// TIA Portal project "MVP" (V18)

(* hardware
DEVICE "S7-1200 station_1"  S7-1200 Station
   slot 0: "Rack_0"  S7-1200 Rack  Rack  V1.0
   slot 1: "PLC_1"  CPU 1214C AC/DC/Rly  6ES7 214-1BG40-0XB0  V4.5
   slot 2: "DI 16/DQ 16x24VDC_1"  6ES7 223-1BL32-0XB0  V2.0
   slot 3: "AI 8x13BIT_1"  6ES7 231-4HF32-0XB0  V2.1
*)

// ===== PLC "PLC_1"  CPU 1214C AC/DC/Rly =====

VAR_GLOBAL   // PLC tag table "Default tag table"
   "VC" AT %Q0.0 : Bool;   // Válvula on/off da entrada do sistema de compressores
   "VT" AT %Q8.1 : Bool;   // Válvula on/off da saída do tanque separador
   "VD1" AT %Q0.2 : Bool;   // Válvula on/off da linha direta (primeira)
   "VD2" AT %Q0.3 : Bool;   // Válvula on/off da linha direta (segunda)
   "C1" AT %Q0.4 : Bool;   // Compressor 1
   "C2" AT %Q0.5 : Bool;   // Compressor 2
   "C3" AT %Q0.6 : Bool;   // Compressor 3
   "LED1" AT %Q0.7 : Bool;   // LED que avisa sobre a pressão no tanque separador
   "LED2" AT %Q1.0 : Bool;   // LED que indica se há alguma operação em curso
   "LE" AT %Q1.1 : Bool;   // LED que indica o estado de Emergência
   "H" AT %Q8.0 : Bool;   // Alarme sonoro
   "BL" AT %I0.0 : Bool;   // Botão Ligar
   "BD" AT %I0.1 : Bool;   // Botão Desligar
   "BE" AT %I0.2 : Bool;   // Botão de Emergência
   "CS1" AT %I0.3 : Bool;   // Chave seletora - Saída 1
   "CS2" AT %I0.4 : Bool;   // Chave seletora - Saída 2
   "P" AT %IW112 : Int;   // Pressão no interior do tanque separador
   "PS" AT %IW114 : Int;   // Pressão na saída do conjunto de compressores
   "PN" AT %IW116 : Int;   // Pressão da linha de abastecimento (nó estendido)
   "T" AT %IW120 : Int;   // Temperatura da linha de abastecimento (nó estendido)
   "BR" AT %I0.5 : Bool;   // Botão Reset
   "BP" AT %I0.6 : Bool;   // Botão Pausa
   "PSF6" AT %IW118 : Int;   // Pressão no tanque de SF6
   "TA" AT %IW122 : Int;   // Temperatura ambiente
   "LED3" AT %Q0.1 : Bool;   // LED que indica início/fim das etapas do MS2
   "LED4" AT %Q8.2 : Bool;   // LED que indica o estado de etapa pausada
   "BU" AT %I0.7 : Bool;   // Botão Retomada (Unpause)
END_VAR

VAR_GLOBAL CONSTANT   // PLC tag table "Default tag table"
   "Pmax" : Real := 8.0;   // Pressão máxima admissível no tanque separador
   "Pmin" : Real := 2.0;   // Pressão mínima admissível no tanque separador
   "PSmax" : Real := 8.0;   // Pressão máxima admissível na saída do conjunto de compressores
   "PSmin" : Real := 2.0;   // Pressão mínima admissível na saída do conjunto de compressores
   "PNmax" : Real := 8.0;   // Pressão máxima admissível no nó estendido
   "PNmin" : Real := 2.0;   // Pressão mínima admissível no nó estendido
   "Lmin" : Real := 4.0;   // Nível mínimo da pressão no tanque separador
   "L2" : Real := 6.0;   // Nível 2 da pressão no tanque separador
   "Tlim" : Real := 4.0;   // Nível mínimo da temperatura no nó estendido
   "Tmax" : Real := 8.0;   // Temperatura máxima admissível no nó estendido
   "Tmin" : Real := 2.0;   // Temperatura mínima admissível no nó estendido
   "gamma" : Real := 0.05;   // Constante para estabelecer um intervalo ao redor de PSF6
   "beta" : Real := 0.05;   // Constante para estabelecer um intervalo ao redor de TA
   "PNlim" : Real := 3.0;   // Nível mínimo da pressão no nó estendido
END_VAR

DATA_BLOCK "Variaveis"   // DB1
{ S7_Optimized_Access := 'TRUE' }
VERSION : 0.1
   VAR
      "Valvulas ON - MS1" : Bool := false;
      n : Int := 0;
      MS1 : Bool := false;
      "Estado anterior - MS1" : Bool := false;
      "Pisca LED1" : Bool := false;
      Inadmissivel : Bool := false;
      Emergencia : Bool := false;
      "Reset delay 1" : Bool := false;
      "Decisao automatica" : Bool := false;
      "VC ON" : Bool := false;
      "Reset delay VC 1" : Bool := false;
      "Aciona compressores" : Bool := false;
      "Reset delay VC 2" : Bool := false;
      "Desliga compressores" : Bool := false;
      MS2 : Bool := false;
      "Estado anterior - MS2" : Bool := false;
      "Aciona VD2" : Bool := false;
      "Transiciona etapa" : Bool := false;
      "VD2 ON" : Bool := false;
      "Desliga VD2" : Bool := false;
      "Tempo estourado - EB" : Bool := false;
      "Tempo estourado - EC" : Bool := false;
      "EB iniciada" : Bool := false;
      "Verifica T igual TA" : Bool := false;
      "Verifica PN e PSF6" : Bool := false;
      "Estado anterior VD2" : Bool := false;
      EB : Bool := false;
      EC : Bool := false;
      "EC iniciada" : Bool := false;
      "Verifica PN e PNlim" : Bool := false;
      "Aciona VC e compressores" : Bool := false;
      "Desliga VC e compressores" : Bool := false;
      "Estado anterior VC e comp" : Bool := false;
      "VC e compressores ON" : Bool := false;
      "Pisca LED3" : Bool := false;
      "Decide etapa" : Bool := false;
      "Etapa pausada" : Bool := false;
      "Etapa retomada" : Bool := false;
      "Pausa OFF" : Bool := false;
      "Estado anterior BP" : Bool := false;
      "BP toggled" : Bool := false;
      "VD1 ON" : Bool := false;
      "Reset delay VD1 VD2 VC" : Bool := false;
      "T inadmissivel" : Bool := false;
      "Pisca LED3 aux" : Bool := false;
      "Realiza EB" : Bool := false;
      "Realiza EC" : Bool := false;
      "LED1 - Piscar" : Bool := false;
      "LED1 - Continuo" : Bool := false;
      "LED1 - Desligar" : Bool := false;
      "Nao desliga BD" : Bool := false;
      "Nao desliga BE" : Bool := false;
      "Nao desliga Inad P" : Bool := false;
      "Nao desliga Inad PS" : Bool := false;
      "Nao desliga Inad PN" : Bool := false;
      "Nao desliga Inad T" : Bool := false;
      "Estado anterior - Emergencia" : Bool := false;
      "Estado anterior - Toggle Inad P" : Bool := false;
      "Estado anterior - Toggle Inad PS" : Bool := false;
      "Estado anterior - Toggle Inad PN" : Bool := false;
      "Estado anterior - Toggle Inad T" : Bool := false;
      "Toggle Emergencia" : Bool := false;
      "Toggle Inad P" : Bool := false;
      "Toggle Inad PS" : Bool := false;
      "Toggle Inad PN" : Bool := false;
      "Toggle Inad T" : Bool := false;
      "Always False" : Bool := false;
      "Reset delay DE" : Bool := false;
      "Reset delay cautela" : Bool := false;
      "Reset delay cautela 2" : Bool := false;
      "Estado anterior - comp MS2" : Bool := false;
      "Estado anterior - desl comp MS2" : Bool := false;
      "Pisca LED2 aux" : Bool := false;
   END_VAR
BEGIN
END_DATA_BLOCK

DATA_BLOCK "Decide LED1 - DB"   // DB19
{ S7_Optimized_Access := 'TRUE' }
VERSION : 0.1
// stored: InstanceOfName Decide LED1 - FB
"Decide LED1 - FB"
BEGIN
END_DATA_BLOCK

// folder: System blocks/Program resources

DATA_BLOCK "Delay 1"   // DB2
{ S7_Optimized_Access := 'TRUE' }
AUTHOR : Simatic
FAMILY : IEC
NAME : IEC_TMR
VERSION : 1.0
// stored: InstanceOfName IEC_TIMER
"IEC_TIMER"
BEGIN
   PT := T#3S;
END_DATA_BLOCK

DATA_BLOCK "Delay VC 1"   // DB3
{ S7_Optimized_Access := 'TRUE' }
AUTHOR : Simatic
FAMILY : IEC
NAME : IEC_TMR
VERSION : 1.0
// stored: InstanceOfName IEC_TIMER
"IEC_TIMER"
BEGIN
   PT := T#5S;
END_DATA_BLOCK

DATA_BLOCK "LED1 ON"   // DB4
{ S7_Optimized_Access := 'TRUE' }
AUTHOR : Simatic
FAMILY : IEC
NAME : IEC_TMR
VERSION : 1.0
// stored: InstanceOfName IEC_TIMER
"IEC_TIMER"
BEGIN
   PT := T#1S;
END_DATA_BLOCK

DATA_BLOCK "LED1 OFF"   // DB5
{ S7_Optimized_Access := 'TRUE' }
AUTHOR : Simatic
FAMILY : IEC
NAME : IEC_TMR
VERSION : 1.0
// stored: InstanceOfName IEC_TIMER
"IEC_TIMER"
BEGIN
   PT := T#1S;
END_DATA_BLOCK

DATA_BLOCK "Reset delay 1"   // DB6
{ S7_Optimized_Access := 'TRUE' }
AUTHOR : Simatic
FAMILY : IEC
NAME : IEC_TMR
VERSION : 1.0
// stored: InstanceOfName IEC_TIMER
"IEC_TIMER"
BEGIN
   PT := T#10MS;
END_DATA_BLOCK

DATA_BLOCK "Reset delay VC 1"   // DB7
{ S7_Optimized_Access := 'TRUE' }
AUTHOR : Simatic
FAMILY : IEC
NAME : IEC_TMR
VERSION : 1.0
// stored: InstanceOfName IEC_TIMER
"IEC_TIMER"
BEGIN
   PT := T#10MS;
END_DATA_BLOCK

DATA_BLOCK "Delay VC 2"   // DB8
{ S7_Optimized_Access := 'TRUE' }
AUTHOR : Simatic
FAMILY : IEC
NAME : IEC_TMR
VERSION : 1.0
// stored: InstanceOfName IEC_TIMER
"IEC_TIMER"
BEGIN
   PT := T#5S;
END_DATA_BLOCK

DATA_BLOCK "Reset delay VC 2"   // DB9
{ S7_Optimized_Access := 'TRUE' }
AUTHOR : Simatic
FAMILY : IEC
NAME : IEC_TMR
VERSION : 1.0
// stored: InstanceOfName IEC_TIMER
"IEC_TIMER"
BEGIN
   PT := T#10MS;
END_DATA_BLOCK

DATA_BLOCK "Contagem EB"   // DB10
{ S7_Optimized_Access := 'TRUE' }
AUTHOR : Simatic
FAMILY : IEC
NAME : IEC_TMR
VERSION : 1.0
// stored: InstanceOfName IEC_TIMER
"IEC_TIMER"
BEGIN
   PT := T#20S;
END_DATA_BLOCK

DATA_BLOCK "Contagem EC"   // DB11
{ S7_Optimized_Access := 'TRUE' }
AUTHOR : Simatic
FAMILY : IEC
NAME : IEC_TMR
VERSION : 1.0
// stored: InstanceOfName IEC_TIMER
"IEC_TIMER"
BEGIN
   PT := T#20S;
END_DATA_BLOCK

DATA_BLOCK "Delay - Decisao etapa"   // DB12
{ S7_Optimized_Access := 'TRUE' }
AUTHOR : Simatic
FAMILY : IEC
NAME : IEC_TMR
VERSION : 1.0
// stored: InstanceOfName IEC_TIMER
"IEC_TIMER"
BEGIN
   PT := T#5S;
END_DATA_BLOCK

DATA_BLOCK "Reset delay DE"   // DB13
{ S7_Optimized_Access := 'TRUE' }
AUTHOR : Simatic
FAMILY : IEC
NAME : IEC_TMR
VERSION : 1.0
// stored: InstanceOfName IEC_TIMER
"IEC_TIMER"
BEGIN
   PT := T#10MS;
END_DATA_BLOCK

DATA_BLOCK "Cautela"   // DB14
{ S7_Optimized_Access := 'TRUE' }
AUTHOR : Simatic
FAMILY : IEC
NAME : IEC_TMR
VERSION : 1.0
// stored: InstanceOfName IEC_TIMER
"IEC_TIMER"
BEGIN
   PT := T#1S;
END_DATA_BLOCK

DATA_BLOCK "LED3 ON"   // DB15
{ S7_Optimized_Access := 'TRUE' }
AUTHOR : Simatic
FAMILY : IEC
NAME : IEC_TMR
VERSION : 1.0
// stored: InstanceOfName IEC_TIMER
"IEC_TIMER"
BEGIN
   PT := T#1S;
END_DATA_BLOCK

DATA_BLOCK "LED3 OFF"   // DB16
{ S7_Optimized_Access := 'TRUE' }
AUTHOR : Simatic
FAMILY : IEC
NAME : IEC_TMR
VERSION : 1.0
// stored: InstanceOfName IEC_TIMER
"IEC_TIMER"
BEGIN
   PT := T#1S;
END_DATA_BLOCK

DATA_BLOCK "Compressores OFF - Inad P"   // DB17
{ S7_Optimized_Access := 'TRUE' }
AUTHOR : Simatic
FAMILY : IEC
NAME : IEC_TMR
VERSION : 1.0
// stored: InstanceOfName IEC_TIMER
"IEC_TIMER"
BEGIN
   PT := T#3S;
END_DATA_BLOCK

DATA_BLOCK "Compressores OFF - BE"   // DB18
{ S7_Optimized_Access := 'TRUE' }
AUTHOR : Simatic
FAMILY : IEC
NAME : IEC_TMR
VERSION : 1.0
// stored: InstanceOfName IEC_TIMER
"IEC_TIMER"
BEGIN
   PT := T#3S;
END_DATA_BLOCK

DATA_BLOCK "Compressores OFF - BD"   // DB20
{ S7_Optimized_Access := 'TRUE' }
AUTHOR : Simatic
FAMILY : IEC
NAME : IEC_TMR
VERSION : 1.0
// stored: InstanceOfName IEC_TIMER
"IEC_TIMER"
BEGIN
   PT := T#3S;
END_DATA_BLOCK

DATA_BLOCK "Compressores OFF - Inad PS"   // DB21
{ S7_Optimized_Access := 'TRUE' }
AUTHOR : Simatic
FAMILY : IEC
NAME : IEC_TMR
VERSION : 1.0
// stored: InstanceOfName IEC_TIMER
"IEC_TIMER"
BEGIN
   PT := T#3S;
END_DATA_BLOCK

DATA_BLOCK "Compressores OFF - Inad PN"   // DB22
{ S7_Optimized_Access := 'TRUE' }
AUTHOR : Simatic
FAMILY : IEC
NAME : IEC_TMR
VERSION : 1.0
// stored: InstanceOfName IEC_TIMER
"IEC_TIMER"
BEGIN
   PT := T#3S;
END_DATA_BLOCK

DATA_BLOCK "Compressores OFF - Inad T"   // DB23
{ S7_Optimized_Access := 'TRUE' }
AUTHOR : Simatic
FAMILY : IEC
NAME : IEC_TMR
VERSION : 1.0
// stored: InstanceOfName IEC_TIMER
"IEC_TIMER"
BEGIN
   PT := T#3S;
END_DATA_BLOCK

DATA_BLOCK "Reset Cautela"   // DB24
{ S7_Optimized_Access := 'TRUE' }
AUTHOR : Simatic
FAMILY : IEC
NAME : IEC_TMR
VERSION : 1.0
// stored: InstanceOfName IEC_TIMER
"IEC_TIMER"
BEGIN
   PT := T#10MS;
END_DATA_BLOCK

DATA_BLOCK "Cautela 2"   // DB25
{ S7_Optimized_Access := 'TRUE' }
AUTHOR : Simatic
FAMILY : IEC
NAME : IEC_TMR
VERSION : 1.0
// stored: InstanceOfName IEC_TIMER
"IEC_TIMER"
BEGIN
   PT := T#20MS;
END_DATA_BLOCK

DATA_BLOCK "Reset Cautela 2"   // DB26
{ S7_Optimized_Access := 'TRUE' }
AUTHOR : Simatic
FAMILY : IEC
NAME : IEC_TMR
VERSION : 1.0
// stored: InstanceOfName IEC_TIMER
"IEC_TIMER"
BEGIN
   PT := T#10MS;
END_DATA_BLOCK

DATA_BLOCK "LED2 ON"   // DB27
{ S7_Optimized_Access := 'TRUE' }
AUTHOR : Simatic
FAMILY : IEC
NAME : IEC_TMR
VERSION : 1.0
// stored: InstanceOfName IEC_TIMER
"IEC_TIMER"
BEGIN
   PT := T#1S;
END_DATA_BLOCK

DATA_BLOCK "LED2 OFF"   // DB28
{ S7_Optimized_Access := 'TRUE' }
AUTHOR : Simatic
FAMILY : IEC
NAME : IEC_TMR
VERSION : 1.0
// stored: InstanceOfName IEC_TIMER
"IEC_TIMER"
BEGIN
   PT := T#1S;
END_DATA_BLOCK

// folder: (top level)

FUNCTION_BLOCK "Decide LED1 - FB"   // FB1, LAD
{ S7_Optimized_Access := 'TRUE' }
VERSION : 0.1
   VAR_INPUT
      P : Real;   // Pressão no tanque separador
   END_VAR
BEGIN

REGION Network 1 (SCL): LED que avisa sobre a pressão no tanque separador
   IF "Variaveis".MS1 = TRUE THEN
       IF #P >= "L2" THEN
           "Variaveis"."LED1 - Continuo" := TRUE;
           "Variaveis"."LED1 - Piscar" := FALSE;
           "Variaveis"."LED1 - Desligar" := FALSE;
       ELSIF #P <= "Lmin" THEN
           "Variaveis"."LED1 - Piscar" := TRUE;
           "Variaveis"."LED1 - Continuo" := FALSE;
           "Variaveis"."LED1 - Desligar" := FALSE;
       ELSE
           "Variaveis"."LED1 - Desligar" := TRUE;
           "Variaveis"."LED1 - Piscar" := FALSE;
           "Variaveis"."LED1 - Continuo" := FALSE;
       END_IF;
   ELSE
       IF #P >= "L2" THEN
           "Variaveis"."LED1 - Continuo" := TRUE;
           "Variaveis"."LED1 - Desligar" := FALSE;
       ELSE
           "Variaveis"."LED1 - Desligar" := TRUE;
           "Variaveis"."LED1 - Continuo" := FALSE;
       END_IF;
   END_IF;
END_REGION
END_FUNCTION_BLOCK

FUNCTION "Aciona valvulas - MS1" : Void   // FC1, LAD
{ S7_Optimized_Access := 'TRUE' }
VERSION : 0.1
BEGIN

REGION Network 1: Válvula on/off da entrada do sistema de compressores
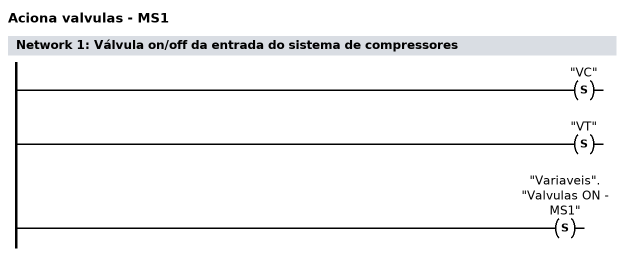
   RUNG wire#powerrail
      S_Coil( "VC" )
   END_RUNG
   RUNG wire#powerrail
      S_Coil( "VT" )
   END_RUNG
   RUNG wire#powerrail
      S_Coil( "Variaveis"."Valvulas ON - MS1" )
   END_RUNG
   // the same network as SCL:
   "VC" := TRUE;
   "VT" := TRUE;
   "Variaveis"."Valvulas ON - MS1" := TRUE;
END_REGION
END_FUNCTION

FUNCTION "Desliga valvulas - MS1" : Void   // FC2, LAD
{ S7_Optimized_Access := 'TRUE' }
VERSION : 0.1
BEGIN

REGION Network 1: Válvula on/off da entrada do sistema de compressores
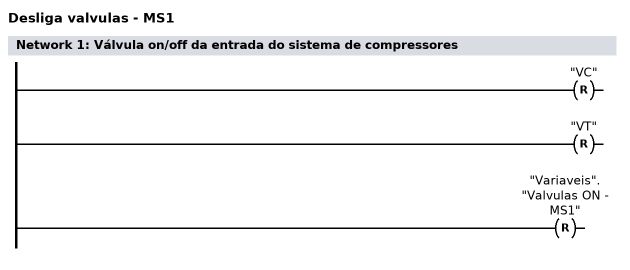
   RUNG wire#powerrail
      R_Coil( "VC" )
   END_RUNG
   RUNG wire#powerrail
      R_Coil( "VT" )
   END_RUNG
   RUNG wire#powerrail
      R_Coil( "Variaveis"."Valvulas ON - MS1" )
   END_RUNG
   // the same network as SCL:
   "VC" := FALSE;
   "VT" := FALSE;
   "Variaveis"."Valvulas ON - MS1" := FALSE;
END_REGION
END_FUNCTION

FUNCTION "Verifica valvulas 1" : Void   // FC3, LAD
{ S7_Optimized_Access := 'TRUE' }
VERSION : 0.1
BEGIN

REGION Network 1
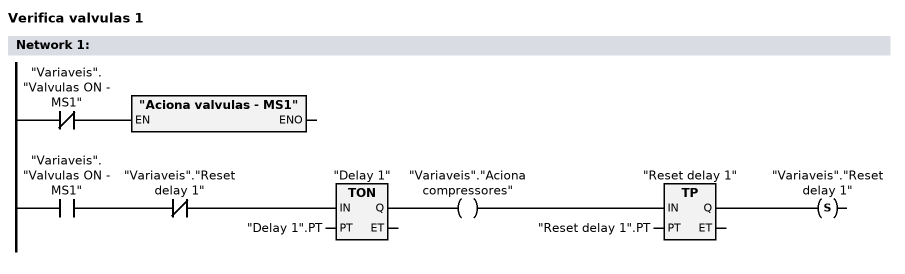
   IF NOT "Variaveis"."Valvulas ON - MS1" THEN "Aciona valvulas - MS1"(); END_IF;
   "Delay 1".TON(IN := "Variaveis"."Valvulas ON - MS1" AND NOT "Variaveis"."Reset delay 1", PT := "Delay 1".PT);
   "Variaveis"."Aciona compressores" := "Delay 1".Q;
   "Reset delay 1".TP(IN := "Delay 1".Q, PT := "Reset delay 1".PT);
   IF "Reset delay 1".Q THEN "Variaveis"."Reset delay 1" := TRUE; END_IF;
END_REGION
END_FUNCTION

FUNCTION "Verifica valvulas 2" : Void   // FC4, LAD
{ S7_Optimized_Access := 'TRUE' }
VERSION : 0.1
BEGIN

REGION Network 1
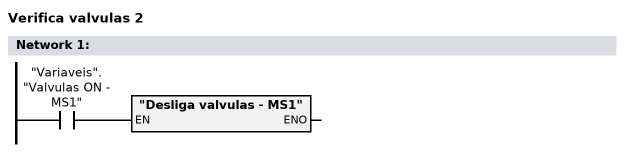
   RUNG wire#powerrail
      Contact( "Variaveis"."Valvulas ON - MS1" )
      "Desliga valvulas - MS1"()
   END_RUNG
   // the same network as SCL:
   IF "Variaveis"."Valvulas ON - MS1" THEN "Desliga valvulas - MS1"(); END_IF;
END_REGION
END_FUNCTION

FUNCTION "Aciona compressores" : Void   // FC5, LAD
{ S7_Optimized_Access := 'TRUE' }
VERSION : 0.1
BEGIN

REGION Network 1: Compressor 1
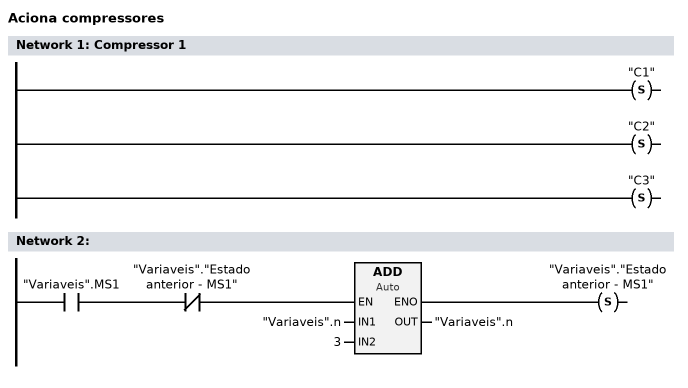
   RUNG wire#powerrail
      S_Coil( "C1" )
   END_RUNG
   RUNG wire#powerrail
      S_Coil( "C2" )
   END_RUNG
   RUNG wire#powerrail
      S_Coil( "C3" )
   END_RUNG
   // the same network as SCL:
   "C1" := TRUE;
   "C2" := TRUE;
   "C3" := TRUE;
END_REGION

REGION Network 2
   RUNG wire#powerrail
      Contact( "Variaveis".MS1 )
      I_Contact( "Variaveis"."Estado anterior - MS1" )
      Add(in1 := "Variaveis".n, in2 := 3, out => "Variaveis".n)
      S_Coil( "Variaveis"."Estado anterior - MS1" )
   END_RUNG
   // the same network as SCL:
   IF "Variaveis".MS1 AND NOT "Variaveis"."Estado anterior - MS1" THEN
       "Variaveis".n := "Variaveis".n + 3;
       "Variaveis"."Estado anterior - MS1" := TRUE;
   END_IF;
END_REGION
END_FUNCTION

FUNCTION "Desliga compressores" : Void   // FC6, LAD
{ S7_Optimized_Access := 'TRUE' }
VERSION : 0.1
BEGIN

REGION Network 1: Compressor 1
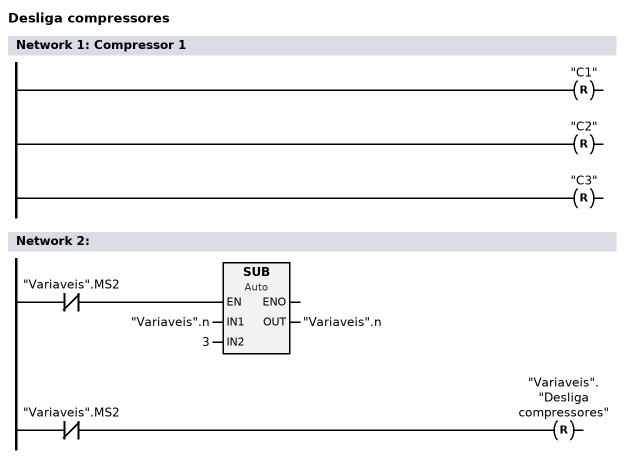
   RUNG wire#powerrail
      R_Coil( "C1" )
   END_RUNG
   RUNG wire#powerrail
      R_Coil( "C2" )
   END_RUNG
   RUNG wire#powerrail
      R_Coil( "C3" )
   END_RUNG
   // the same network as SCL:
   "C1" := FALSE;
   "C2" := FALSE;
   "C3" := FALSE;
END_REGION

REGION Network 2
   RUNG wire#powerrail
      I_Contact( "Variaveis".MS2 )
      Sub(in1 := "Variaveis".n, in2 := 3, out => "Variaveis".n)
   END_RUNG
   RUNG wire#powerrail
      I_Contact( "Variaveis".MS2 )
      R_Coil( "Variaveis"."Desliga compressores" )
   END_RUNG
   // the same network as SCL:
   IF NOT "Variaveis".MS2 THEN
       "Variaveis".n := "Variaveis".n - 3;
       "Variaveis"."Desliga compressores" := FALSE;
   END_IF;
END_REGION
END_FUNCTION

FUNCTION "Verifica compressores" : Void   // FC7, LAD
{ S7_Optimized_Access := 'TRUE' }
VERSION : 0.1
BEGIN

REGION Network 1
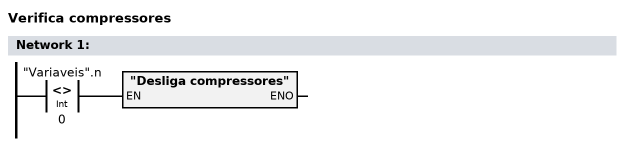
   RUNG wire#powerrail
      { S7_Templates := "SrcType := Int" } NE_Contact(in1 := "Variaveis".n, in2 := 0)
      "Desliga compressores"()
   END_RUNG
   // the same network as SCL:
   IF "Variaveis".n <> 0 THEN "Desliga compressores"(); END_IF;
END_REGION
END_FUNCTION

FUNCTION "Finaliza operacao - MS1" : Void   // FC8, LAD
{ S7_Optimized_Access := 'TRUE' }
VERSION : 0.1
BEGIN

REGION Network 1
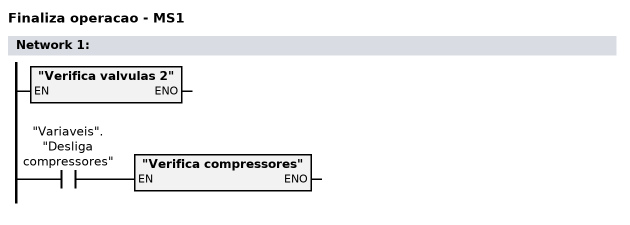
   RUNG wire#powerrail
      "Verifica valvulas 2"()
   END_RUNG
   RUNG wire#powerrail
      Contact( "Variaveis"."Desliga compressores" )
      "Verifica compressores"()
   END_RUNG
   // the same network as SCL:
   "Verifica valvulas 2"();
   IF "Variaveis"."Desliga compressores" THEN "Verifica compressores"(); END_IF;
END_REGION
END_FUNCTION

FUNCTION "MS1 - Operacao iniciada" : Void   // FC9, LAD
{ S7_Optimized_Access := 'TRUE' }
VERSION : 0.1
BEGIN

REGION Network 1
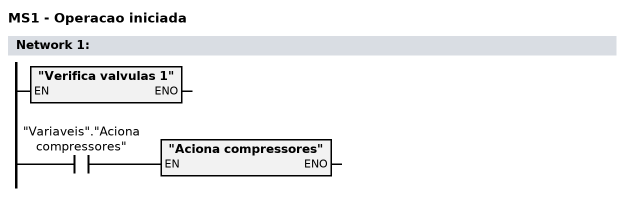
   RUNG wire#powerrail
      "Verifica valvulas 1"()
   END_RUNG
   RUNG wire#powerrail
      Contact( "Variaveis"."Aciona compressores" )
      "Aciona compressores"()
   END_RUNG
   // the same network as SCL:
   "Verifica valvulas 1"();
   IF "Variaveis"."Aciona compressores" THEN "Aciona compressores"(); END_IF;
END_REGION
END_FUNCTION

FUNCTION "MS1 - Operacao finalizada" : Void   // FC10, LAD
{ S7_Optimized_Access := 'TRUE' }
VERSION : 0.1
BEGIN

REGION Network 1
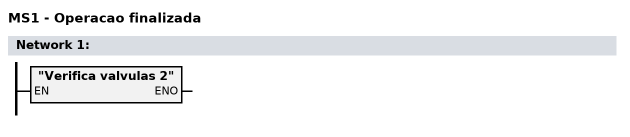
   RUNG wire#powerrail
      "Verifica valvulas 2"()
   END_RUNG
   // the same network as SCL:
   "Verifica valvulas 2"();
END_REGION
END_FUNCTION

FUNCTION "OPERACAO - MS1" : Void   // FC11, LAD
{ S7_Optimized_Access := 'TRUE' }
VERSION : 0.1
   VAR_TEMP   // added for the SCL form of the ladder/FBD networks
      _w1 : Bool;
   END_VAR
BEGIN

REGION Network 1: LED que indica se há alguma operação em curso
   // Em operação
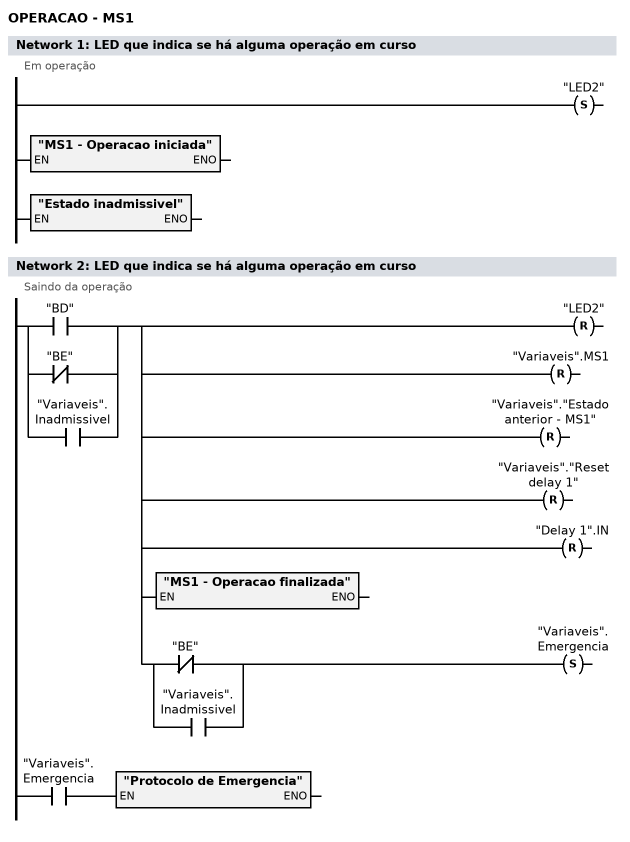
   RUNG wire#powerrail
      S_Coil( "LED2" )
   END_RUNG
   RUNG wire#powerrail
      "MS1 - Operacao iniciada"()
   END_RUNG
   RUNG wire#powerrail
      "Estado inadmissivel"()
   END_RUNG
   // the same network as SCL:
   "LED2" := TRUE;
   "MS1 - Operacao iniciada"();
   "Estado inadmissivel"();
END_REGION

REGION Network 2: LED que indica se há alguma operação em curso
   // Saindo da operação
   RUNG wire#powerrail
      Contact( "BD" )
      wire#w1
      R_Coil( "LED2" )
   END_RUNG
   RUNG wire#powerrail
      I_Contact( "BE" )
   END_RUNG wire#w1
   RUNG wire#powerrail
      Contact( "Variaveis".Inadmissivel )
   END_RUNG wire#w1
   RUNG wire#w1
      R_Coil( "Variaveis".MS1 )
   END_RUNG
   RUNG wire#w1
      R_Coil( "Variaveis"."Estado anterior - MS1" )
   END_RUNG
   RUNG wire#w1
      R_Coil( "Variaveis"."Reset delay 1" )
   END_RUNG
   RUNG wire#w1
      R_Coil( "Delay 1".IN )
   END_RUNG
   RUNG wire#w1
      "MS1 - Operacao finalizada"()
   END_RUNG
   RUNG wire#w1
      I_Contact( "BE" )
      wire#w2
      S_Coil( "Variaveis".Emergencia )
   END_RUNG
   RUNG wire#w1
      Contact( "Variaveis".Inadmissivel )
   END_RUNG wire#w2
   RUNG wire#powerrail
      Contact( "Variaveis".Emergencia )
      "Protocolo de Emergencia"()
   END_RUNG
   // the same network as SCL:
   #_w1 := "BD" OR NOT "BE" OR "Variaveis".Inadmissivel;
   IF #_w1 THEN
       "LED2" := FALSE;
       "Variaveis".MS1 := FALSE;
       "Variaveis"."Estado anterior - MS1" := FALSE;
       "Variaveis"."Reset delay 1" := FALSE;
       "Delay 1".IN := FALSE;
       "MS1 - Operacao finalizada"();
   END_IF;
   IF #_w1 AND (NOT "BE" OR "Variaveis".Inadmissivel) THEN "Variaveis".Emergencia := TRUE; END_IF;
   IF "Variaveis".Emergencia THEN "Protocolo de Emergencia"(); END_IF;
END_REGION
END_FUNCTION

FUNCTION "Pisca LED2" : Void   // FC12, LAD
{ S7_Optimized_Access := 'TRUE' }
VERSION : 0.1
   VAR_TEMP   // added for the SCL form of the ladder/FBD networks
      _w1 : Bool;
   END_VAR
BEGIN

REGION Network 1: LED que indica início/fim das etapas do MS2
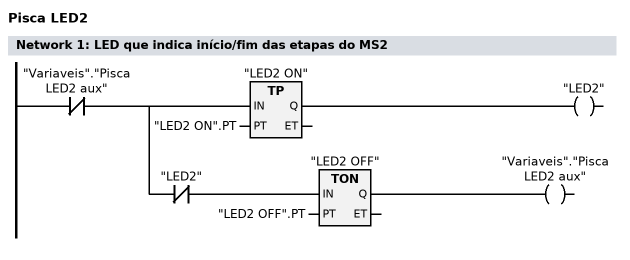
   #_w1 := NOT "Variaveis"."Pisca LED2 aux";
   "LED2 ON".TP(IN := #_w1, PT := "LED2 ON".PT);
   "LED2" := "LED2 ON".Q;
   "LED2 OFF".TON(IN := #_w1 AND NOT "LED2", PT := "LED2 OFF".PT);
   "Variaveis"."Pisca LED2 aux" := "LED2 OFF".Q;
END_REGION
END_FUNCTION

FUNCTION "Obtem pressao P" : Void   // FC13, LAD
{ S7_Optimized_Access := 'TRUE' }
VERSION : 0.1
   VAR_OUTPUT
      P : Real;   // Pressão obtida
   END_VAR
   VAR_TEMP
      "Pressao normalizada" : Real;   // Pressão normalizada
   END_VAR
BEGIN

REGION Network 1
   // Normalização do valor de pressão lido do transmissor
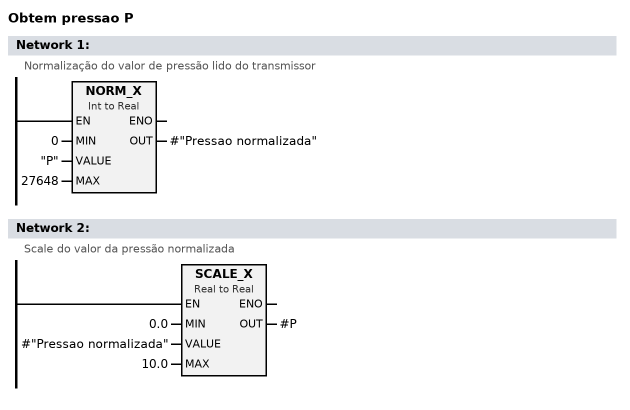
   RUNG wire#powerrail
      { S7_Templates := "[SrcType := Int, DestType := Real]" } Normalize(min := 0, value := "P", max := 27648, out => #"Pressao normalizada")
   END_RUNG
   // the same network as SCL:
   #"Pressao normalizada" := NORM_X(MIN := 0, VALUE := "P", MAX := 27648);
END_REGION

REGION Network 2
   // Scale do valor da pressão normalizada
   RUNG wire#powerrail
      { S7_Templates := "[SrcType := Real, DestType := Real]" } Scale(min := 0.0, value := #"Pressao normalizada", max := 10.0, out => #P)
   END_RUNG
   // the same network as SCL:
   #P := SCALE_X(MIN := 0.0, VALUE := #"Pressao normalizada", MAX := 10.0);
END_REGION
END_FUNCTION

FUNCTION "Estado inadmissivel" : Void   // FC14, LAD
{ S7_Optimized_Access := 'TRUE' }
VERSION : 0.1
   VAR_TEMP
      P : Real;   // Pressão P
      PS : Real;   // Pressão PS
      PN : Real;   // Pressão PN
   END_VAR
BEGIN

REGION Network 1
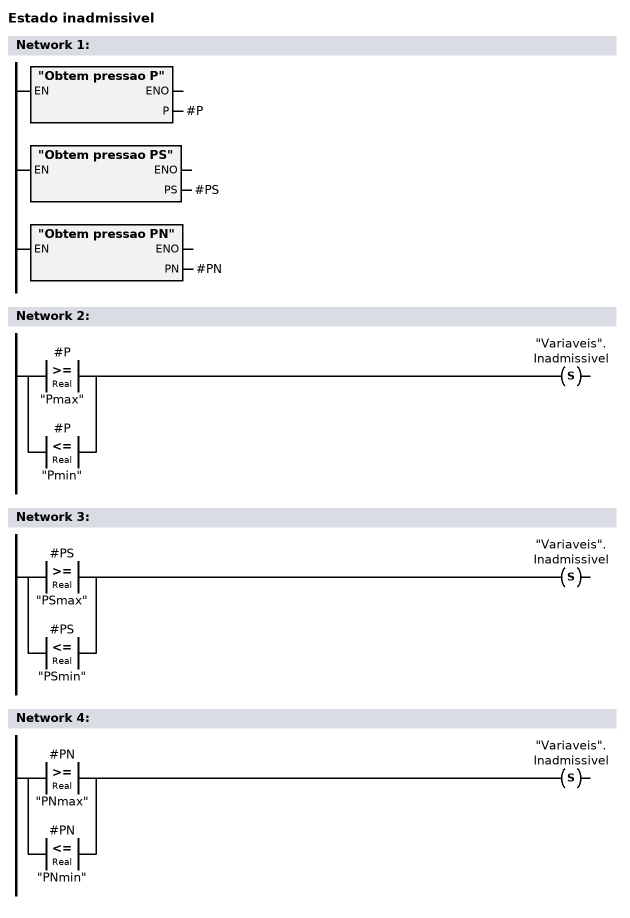
   RUNG wire#powerrail
      "Obtem pressao P"(P => #P)
   END_RUNG
   RUNG wire#powerrail
      "Obtem pressao PS"(PS => #PS)
   END_RUNG
   RUNG wire#powerrail
      "Obtem pressao PN"(PN => #PN)
   END_RUNG
   // the same network as SCL:
   "Obtem pressao P"(P => #P);
   "Obtem pressao PS"(PS => #PS);
   "Obtem pressao PN"(PN => #PN);
END_REGION

REGION Network 2
   RUNG wire#powerrail
      { S7_Templates := "SrcType := Real" } GE_Contact(in1 := #P, in2 := "Pmax")
      wire#w1
      S_Coil( "Variaveis".Inadmissivel )
   END_RUNG
   RUNG wire#powerrail
      { S7_Templates := "SrcType := Real" } LE_Contact(in1 := #P, in2 := "Pmin")
   END_RUNG wire#w1
   // the same network as SCL:
   IF (#P >= "Pmax") OR (#P <= "Pmin") THEN "Variaveis".Inadmissivel := TRUE; END_IF;
END_REGION

REGION Network 3
   RUNG wire#powerrail
      { S7_Templates := "SrcType := Real" } GE_Contact(in1 := #PS, in2 := "PSmax")
      wire#w1
      S_Coil( "Variaveis".Inadmissivel )
   END_RUNG
   RUNG wire#powerrail
      { S7_Templates := "SrcType := Real" } LE_Contact(in1 := #PS, in2 := "PSmin")
   END_RUNG wire#w1
   // the same network as SCL:
   IF (#PS >= "PSmax") OR (#PS <= "PSmin") THEN "Variaveis".Inadmissivel := TRUE; END_IF;
END_REGION

REGION Network 4
   RUNG wire#powerrail
      { S7_Templates := "SrcType := Real" } GE_Contact(in1 := #PN, in2 := "PNmax")
      wire#w1
      S_Coil( "Variaveis".Inadmissivel )
   END_RUNG
   RUNG wire#powerrail
      { S7_Templates := "SrcType := Real" } LE_Contact(in1 := #PN, in2 := "PNmin")
   END_RUNG wire#w1
   // the same network as SCL:
   IF (#PN >= "PNmax") OR (#PN <= "PNmin") THEN "Variaveis".Inadmissivel := TRUE; END_IF;
END_REGION
END_FUNCTION

FUNCTION "Obtem pressao PS" : Void   // FC15, LAD
{ S7_Optimized_Access := 'TRUE' }
VERSION : 0.1
   VAR_OUTPUT
      PS : Real;   // Pressão obtida
   END_VAR
   VAR_TEMP
      "Pressao normalizada" : Real;   // Pressão normalizada
   END_VAR
BEGIN

REGION Network 1
   // Normalização do valor de pressão lido do transmissor
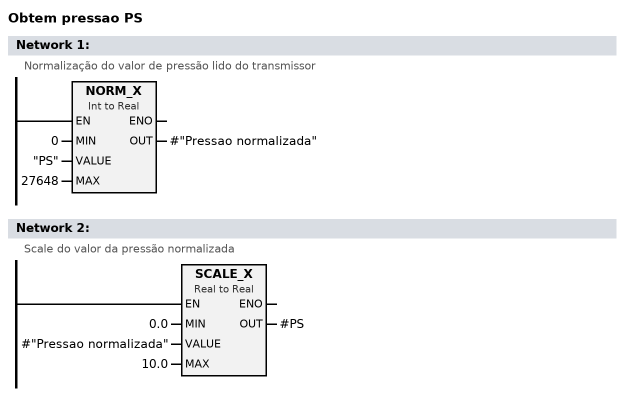
   RUNG wire#powerrail
      { S7_Templates := "[SrcType := Int, DestType := Real]" } Normalize(min := 0, value := "PS", max := 27648, out => #"Pressao normalizada")
   END_RUNG
   // the same network as SCL:
   #"Pressao normalizada" := NORM_X(MIN := 0, VALUE := "PS", MAX := 27648);
END_REGION

REGION Network 2
   // Scale do valor da pressão normalizada
   RUNG wire#powerrail
      { S7_Templates := "[SrcType := Real, DestType := Real]" } Scale(min := 0.0, value := #"Pressao normalizada", max := 10.0, out => #PS)
   END_RUNG
   // the same network as SCL:
   #PS := SCALE_X(MIN := 0.0, VALUE := #"Pressao normalizada", MAX := 10.0);
END_REGION
END_FUNCTION

FUNCTION "Obtem pressao PN" : Void   // FC16, LAD
{ S7_Optimized_Access := 'TRUE' }
VERSION : 0.1
   VAR_OUTPUT
      PN : Real;   // Pressão obtida
   END_VAR
   VAR_TEMP
      "Pressao normalizada" : Real;   // Pressão normalizada
   END_VAR
BEGIN

REGION Network 1
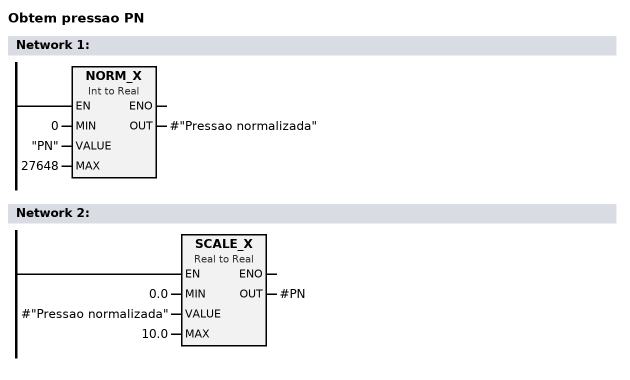
   RUNG wire#powerrail
      { S7_Templates := "[SrcType := Int, DestType := Real]" } Normalize(min := 0, value := "PN", max := 27648, out => #"Pressao normalizada")
   END_RUNG
   // the same network as SCL:
   #"Pressao normalizada" := NORM_X(MIN := 0, VALUE := "PN", MAX := 27648);
END_REGION

REGION Network 2
   RUNG wire#powerrail
      { S7_Templates := "[SrcType := Real, DestType := Real]" } Scale(min := 0.0, value := #"Pressao normalizada", max := 10.0, out => #PN)
   END_RUNG
   // the same network as SCL:
   #PN := SCALE_X(MIN := 0.0, VALUE := #"Pressao normalizada", MAX := 10.0);
END_REGION
END_FUNCTION

FUNCTION "Protocolo de Emergencia" : Void   // FC17, LAD
{ S7_Optimized_Access := 'TRUE' }
VERSION : 0.1
BEGIN

REGION Network 1: LED que indica o estado de Emergência
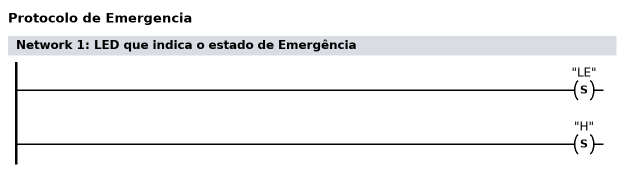
   RUNG wire#powerrail
      S_Coil( "LE" )
   END_RUNG
   RUNG wire#powerrail
      S_Coil( "H" )
   END_RUNG
   // the same network as SCL:
   "LE" := TRUE;
   "H" := TRUE;
END_REGION
END_FUNCTION

FUNCTION "Logica conjunta" : Void   // FC18, LAD
{ S7_Optimized_Access := 'TRUE' }
VERSION : 0.1
   VAR_TEMP
      P : Real;
      PS : Real;
      PN : Real;
      T : Real;
   END_VAR
BEGIN

REGION Network 1
   // Chave seletora na posição 1
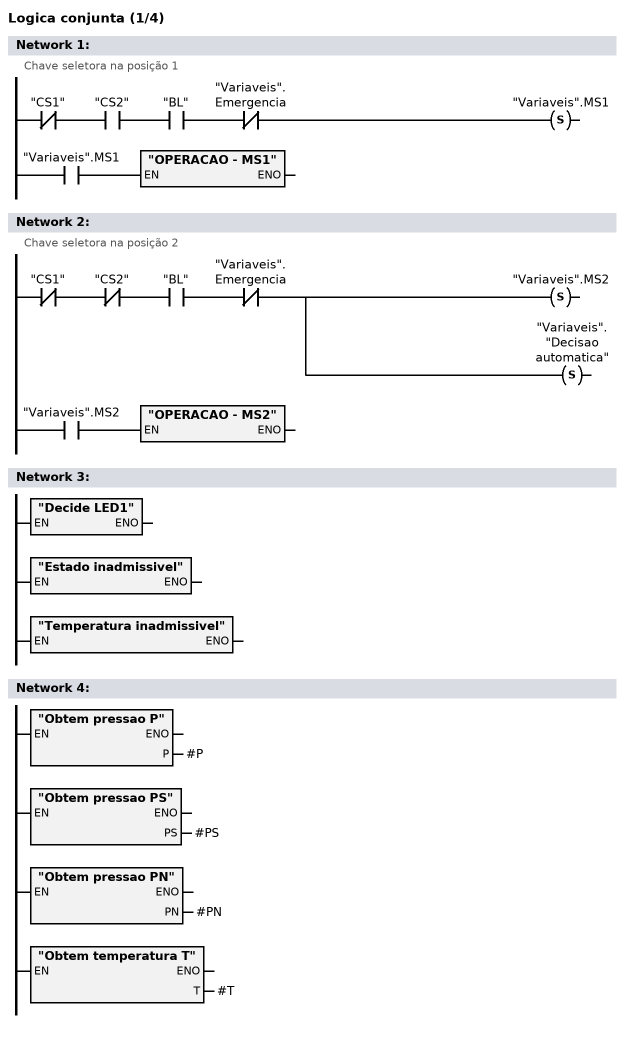
   RUNG wire#powerrail
      I_Contact( "CS1" )
      Contact( "CS2" )
      Contact( "BL" )
      I_Contact( "Variaveis".Emergencia )
      S_Coil( "Variaveis".MS1 )
   END_RUNG
   RUNG wire#powerrail
      Contact( "Variaveis".MS1 )
      "OPERACAO - MS1"()
   END_RUNG
   // the same network as SCL:
   IF NOT "CS1" AND "CS2" AND "BL" AND NOT "Variaveis".Emergencia THEN "Variaveis".MS1 := TRUE; END_IF;
   IF "Variaveis".MS1 THEN "OPERACAO - MS1"(); END_IF;
END_REGION

REGION Network 2
   // Chave seletora na posição 2
   RUNG wire#powerrail
      I_Contact( "CS1" )
      I_Contact( "CS2" )
      Contact( "BL" )
      I_Contact( "Variaveis".Emergencia )
      wire#w1
      S_Coil( "Variaveis".MS2 )
   END_RUNG
   RUNG wire#w1
      S_Coil( "Variaveis"."Decisao automatica" )
   END_RUNG
   RUNG wire#powerrail
      Contact( "Variaveis".MS2 )
      "OPERACAO - MS2"()
   END_RUNG
   // the same network as SCL:
   IF NOT "CS1" AND NOT "CS2" AND "BL" AND NOT "Variaveis".Emergencia THEN
       "Variaveis".MS2 := TRUE;
       "Variaveis"."Decisao automatica" := TRUE;
   END_IF;
   IF "Variaveis".MS2 THEN "OPERACAO - MS2"(); END_IF;
END_REGION

REGION Network 3
   RUNG wire#powerrail
      "Decide LED1"()
   END_RUNG
   RUNG wire#powerrail
      "Estado inadmissivel"()
   END_RUNG
   RUNG wire#powerrail
      "Temperatura inadmissivel"()
   END_RUNG
   // the same network as SCL:
   "Decide LED1"();
   "Estado inadmissivel"();
   "Temperatura inadmissivel"();
END_REGION

REGION Network 4
   RUNG wire#powerrail
      "Obtem pressao P"(P => #P)
   END_RUNG
   RUNG wire#powerrail
      "Obtem pressao PS"(PS => #PS)
   END_RUNG
   RUNG wire#powerrail
      "Obtem pressao PN"(PN => #PN)
   END_RUNG
   RUNG wire#powerrail
      "Obtem temperatura T"(T => #T)
   END_RUNG
   // the same network as SCL:
   "Obtem pressao P"(P => #P);
   "Obtem pressao PS"(PS => #PS);
   "Obtem pressao PN"(PN => #PN);
   "Obtem temperatura T"(T => #T);
END_REGION

REGION Network 5
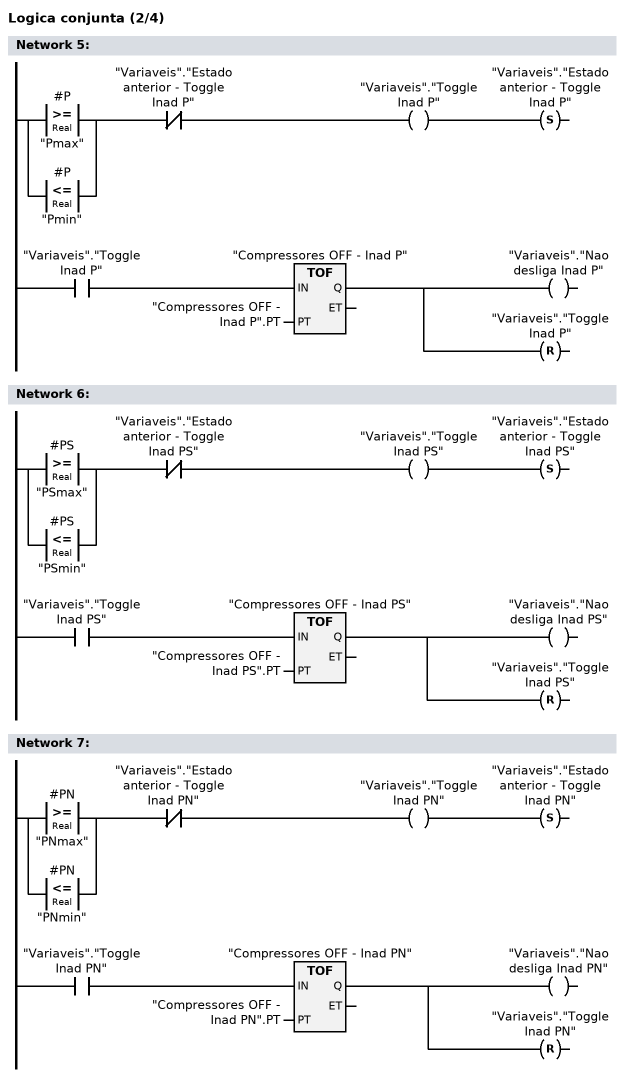
   "Variaveis"."Toggle Inad P" := ((#P >= "Pmax") OR (#P <= "Pmin")) AND NOT "Variaveis"."Estado anterior - Toggle Inad P";
   IF "Variaveis"."Toggle Inad P" THEN "Variaveis"."Estado anterior - Toggle Inad P" := TRUE; END_IF;
   "Compressores OFF - Inad P".TOF(IN := "Variaveis"."Toggle Inad P", PT := "Compressores OFF - Inad P".PT);
   "Variaveis"."Nao desliga Inad P" := "Compressores OFF - Inad P".Q;
   IF "Compressores OFF - Inad P".Q THEN "Variaveis"."Toggle Inad P" := FALSE; END_IF;
END_REGION

REGION Network 6
   "Variaveis"."Toggle Inad PS" := ((#PS >= "PSmax") OR (#PS <= "PSmin")) AND NOT "Variaveis"."Estado anterior - Toggle Inad PS";
   IF "Variaveis"."Toggle Inad PS" THEN "Variaveis"."Estado anterior - Toggle Inad PS" := TRUE; END_IF;
   "Compressores OFF - Inad PS".TOF(IN := "Variaveis"."Toggle Inad PS", PT := "Compressores OFF - Inad PS".PT);
   "Variaveis"."Nao desliga Inad PS" := "Compressores OFF - Inad PS".Q;
   IF "Compressores OFF - Inad PS".Q THEN "Variaveis"."Toggle Inad PS" := FALSE; END_IF;
END_REGION

REGION Network 7
   "Variaveis"."Toggle Inad PN" := ((#PN >= "PNmax") OR (#PN <= "PNmin")) AND NOT "Variaveis"."Estado anterior - Toggle Inad PN";
   IF "Variaveis"."Toggle Inad PN" THEN "Variaveis"."Estado anterior - Toggle Inad PN" := TRUE; END_IF;
   "Compressores OFF - Inad PN".TOF(IN := "Variaveis"."Toggle Inad PN", PT := "Compressores OFF - Inad PN".PT);
   "Variaveis"."Nao desliga Inad PN" := "Compressores OFF - Inad PN".Q;
   IF "Compressores OFF - Inad PN".Q THEN "Variaveis"."Toggle Inad PN" := FALSE; END_IF;
END_REGION

REGION Network 8
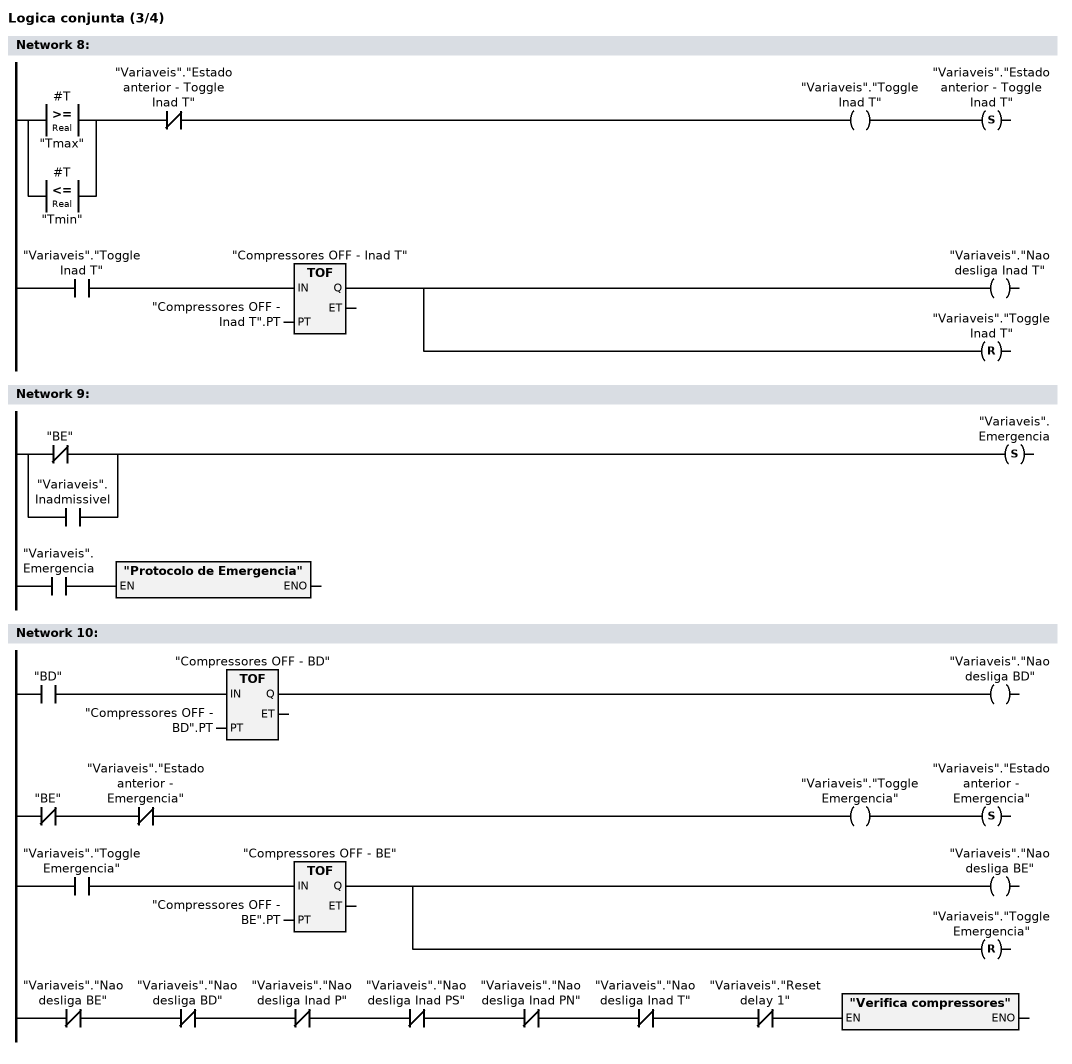
   "Variaveis"."Toggle Inad T" := ((#T >= "Tmax") OR (#T <= "Tmin")) AND NOT "Variaveis"."Estado anterior - Toggle Inad T";
   IF "Variaveis"."Toggle Inad T" THEN "Variaveis"."Estado anterior - Toggle Inad T" := TRUE; END_IF;
   "Compressores OFF - Inad T".TOF(IN := "Variaveis"."Toggle Inad T", PT := "Compressores OFF - Inad T".PT);
   "Variaveis"."Nao desliga Inad T" := "Compressores OFF - Inad T".Q;
   IF "Compressores OFF - Inad T".Q THEN "Variaveis"."Toggle Inad T" := FALSE; END_IF;
END_REGION

REGION Network 9
   RUNG wire#powerrail
      I_Contact( "BE" )
      wire#w1
      S_Coil( "Variaveis".Emergencia )
   END_RUNG
   RUNG wire#powerrail
      Contact( "Variaveis".Inadmissivel )
   END_RUNG wire#w1
   RUNG wire#powerrail
      Contact( "Variaveis".Emergencia )
      "Protocolo de Emergencia"()
   END_RUNG
   // the same network as SCL:
   IF NOT "BE" OR "Variaveis".Inadmissivel THEN "Variaveis".Emergencia := TRUE; END_IF;
   IF "Variaveis".Emergencia THEN "Protocolo de Emergencia"(); END_IF;
END_REGION

REGION Network 10
   "Compressores OFF - BD".TOF(IN := "BD", PT := "Compressores OFF - BD".PT);
   "Variaveis"."Nao desliga BD" := "Compressores OFF - BD".Q;
   "Variaveis"."Toggle Emergencia" := NOT "BE" AND NOT "Variaveis"."Estado anterior - Emergencia";
   IF "Variaveis"."Toggle Emergencia" THEN "Variaveis"."Estado anterior - Emergencia" := TRUE; END_IF;
   "Compressores OFF - BE".TOF(IN := "Variaveis"."Toggle Emergencia", PT := "Compressores OFF - BE".PT);
   "Variaveis"."Nao desliga BE" := "Compressores OFF - BE".Q;
   IF "Compressores OFF - BE".Q THEN "Variaveis"."Toggle Emergencia" := FALSE; END_IF;
   IF NOT "Variaveis"."Nao desliga BE" AND NOT "Variaveis"."Nao desliga BD" AND NOT "Variaveis"."Nao desliga Inad P" AND NOT "Variaveis"."Nao desliga Inad PS" AND NOT "Variaveis"."Nao desliga Inad PN" AND NOT "Variaveis"."Nao desliga Inad T" AND NOT "Variaveis"."Reset delay 1" THEN
       "Verifica compressores"();
   END_IF;
END_REGION

REGION Network 11
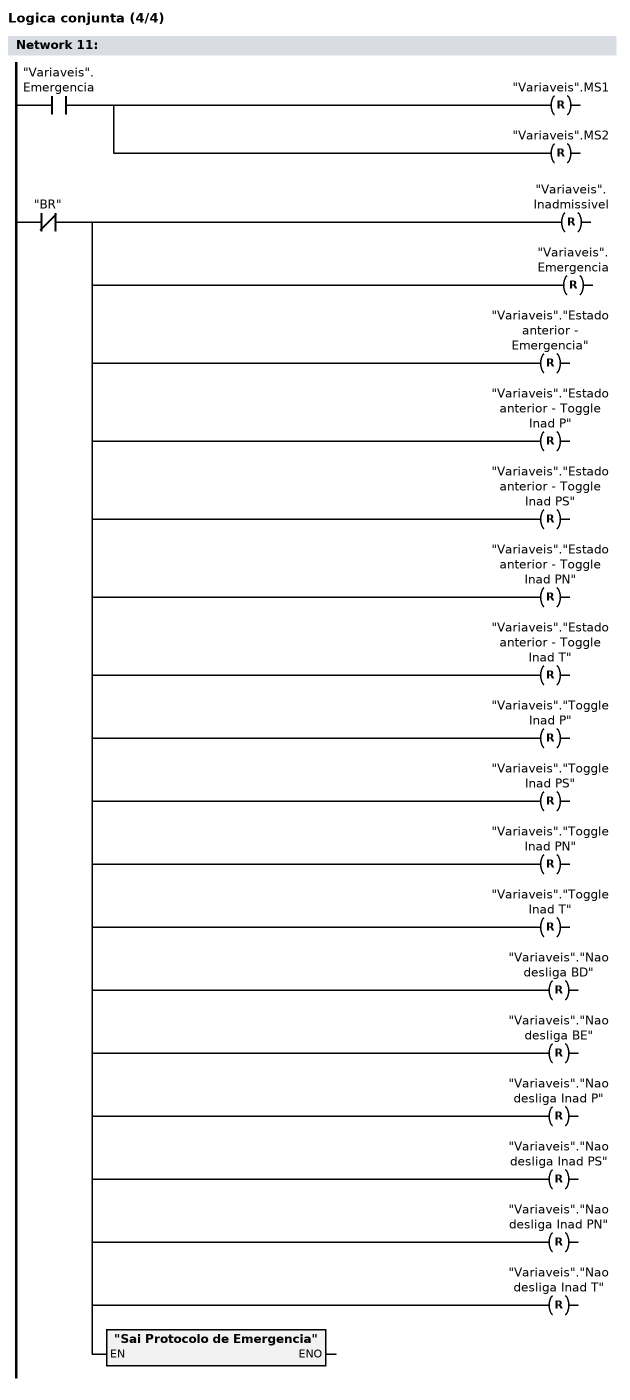
   RUNG wire#powerrail
      Contact( "Variaveis".Emergencia )
      wire#w1
      R_Coil( "Variaveis".MS1 )
   END_RUNG
   RUNG wire#w1
      R_Coil( "Variaveis".MS2 )
   END_RUNG
   RUNG wire#powerrail
      I_Contact( "BR" )
      wire#w2
      R_Coil( "Variaveis".Inadmissivel )
   END_RUNG
   RUNG wire#w2
      R_Coil( "Variaveis".Emergencia )
   END_RUNG
   RUNG wire#w2
      R_Coil( "Variaveis"."Estado anterior - Emergencia" )
   END_RUNG
   RUNG wire#w2
      R_Coil( "Variaveis"."Estado anterior - Toggle Inad P" )
   END_RUNG
   RUNG wire#w2
      R_Coil( "Variaveis"."Estado anterior - Toggle Inad PS" )
   END_RUNG
   RUNG wire#w2
      R_Coil( "Variaveis"."Estado anterior - Toggle Inad PN" )
   END_RUNG
   RUNG wire#w2
      R_Coil( "Variaveis"."Estado anterior - Toggle Inad T" )
   END_RUNG
   RUNG wire#w2
      R_Coil( "Variaveis"."Toggle Inad P" )
   END_RUNG
   RUNG wire#w2
      R_Coil( "Variaveis"."Toggle Inad PS" )
   END_RUNG
   RUNG wire#w2
      R_Coil( "Variaveis"."Toggle Inad PN" )
   END_RUNG
   RUNG wire#w2
      R_Coil( "Variaveis"."Toggle Inad T" )
   END_RUNG
   RUNG wire#w2
      R_Coil( "Variaveis"."Nao desliga BD" )
   END_RUNG
   RUNG wire#w2
      R_Coil( "Variaveis"."Nao desliga BE" )
   END_RUNG
   RUNG wire#w2
      R_Coil( "Variaveis"."Nao desliga Inad P" )
   END_RUNG
   RUNG wire#w2
      R_Coil( "Variaveis"."Nao desliga Inad PS" )
   END_RUNG
   RUNG wire#w2
      R_Coil( "Variaveis"."Nao desliga Inad PN" )
   END_RUNG
   RUNG wire#w2
      R_Coil( "Variaveis"."Nao desliga Inad T" )
   END_RUNG
   RUNG wire#w2
      "Sai Protocolo de Emergencia"()
   END_RUNG
   // the same network as SCL:
   IF "Variaveis".Emergencia THEN
       "Variaveis".MS1 := FALSE;
       "Variaveis".MS2 := FALSE;
   END_IF;
   IF NOT "BR" THEN
       "Variaveis".Inadmissivel := FALSE;
       "Variaveis".Emergencia := FALSE;
       "Variaveis"."Estado anterior - Emergencia" := FALSE;
       "Variaveis"."Estado anterior - Toggle Inad P" := FALSE;
       "Variaveis"."Estado anterior - Toggle Inad PS" := FALSE;
       "Variaveis"."Estado anterior - Toggle Inad PN" := FALSE;
       "Variaveis"."Estado anterior - Toggle Inad T" := FALSE;
       "Variaveis"."Toggle Inad P" := FALSE;
       "Variaveis"."Toggle Inad PS" := FALSE;
       "Variaveis"."Toggle Inad PN" := FALSE;
       "Variaveis"."Toggle Inad T" := FALSE;
       "Variaveis"."Nao desliga BD" := FALSE;
       "Variaveis"."Nao desliga BE" := FALSE;
       "Variaveis"."Nao desliga Inad P" := FALSE;
       "Variaveis"."Nao desliga Inad PS" := FALSE;
       "Variaveis"."Nao desliga Inad PN" := FALSE;
       "Variaveis"."Nao desliga Inad T" := FALSE;
       "Sai Protocolo de Emergencia"();
   END_IF;
END_REGION
END_FUNCTION

FUNCTION "Decide LED1" : Void   // FC19, LAD
{ S7_Optimized_Access := 'TRUE' }
VERSION : 0.1
   VAR_TEMP
      P : Real;   // Pressao obtida no tanque separador
   END_VAR
   VAR_TEMP   // added for the SCL form of the ladder/FBD networks
      _w1 : Bool;
   END_VAR
BEGIN

REGION Network 1
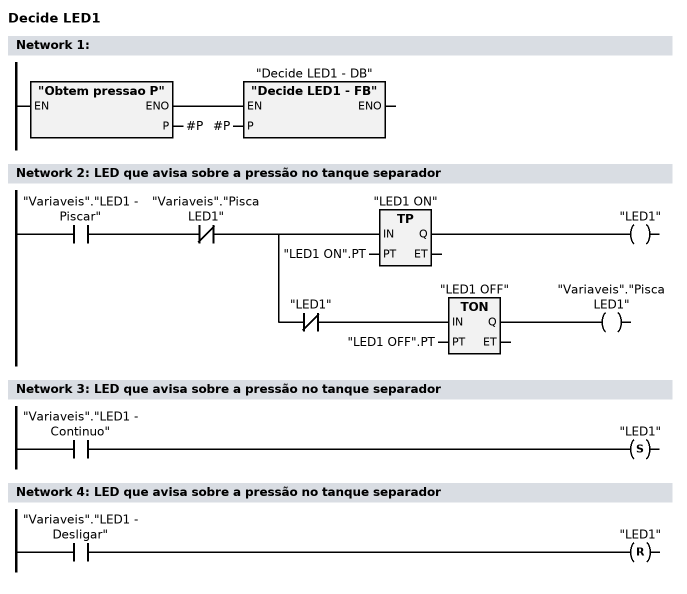
   RUNG wire#powerrail
      "Obtem pressao P"(P => #P)
      "Decide LED1 - DB"(P := #P)
   END_RUNG
   // the same network as SCL:
   "Obtem pressao P"(P => #P, ENO => #_w1);
   IF #_w1 THEN
       "Decide LED1 - DB"(P := #P);   // "Decide LED1 - FB"
   END_IF;
END_REGION

REGION Network 2: LED que avisa sobre a pressão no tanque separador
   #_w1 := "Variaveis"."LED1 - Piscar" AND NOT "Variaveis"."Pisca LED1";
   "LED1 ON".TP(IN := #_w1, PT := "LED1 ON".PT);
   "LED1" := "LED1 ON".Q;
   "LED1 OFF".TON(IN := #_w1 AND NOT "LED1", PT := "LED1 OFF".PT);
   "Variaveis"."Pisca LED1" := "LED1 OFF".Q;
END_REGION

REGION Network 3: LED que avisa sobre a pressão no tanque separador
   RUNG wire#powerrail
      Contact( "Variaveis"."LED1 - Continuo" )
      S_Coil( "LED1" )
   END_RUNG
   // the same network as SCL:
   IF "Variaveis"."LED1 - Continuo" THEN "LED1" := TRUE; END_IF;
END_REGION

REGION Network 4: LED que avisa sobre a pressão no tanque separador
   RUNG wire#powerrail
      Contact( "Variaveis"."LED1 - Desligar" )
      R_Coil( "LED1" )
   END_RUNG
   // the same network as SCL:
   IF "Variaveis"."LED1 - Desligar" THEN "LED1" := FALSE; END_IF;
END_REGION
END_FUNCTION

FUNCTION "Sai Protocolo de Emergencia" : Void   // FC20, LAD
{ S7_Optimized_Access := 'TRUE' }
VERSION : 0.1
BEGIN

REGION Network 1: LED que indica o estado de Emergência
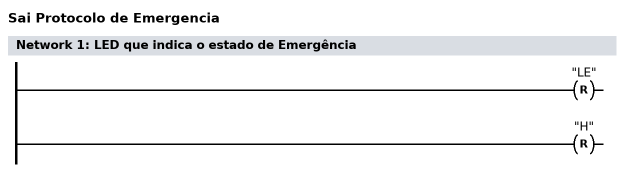
   RUNG wire#powerrail
      R_Coil( "LE" )
   END_RUNG
   RUNG wire#powerrail
      R_Coil( "H" )
   END_RUNG
   // the same network as SCL:
   "LE" := FALSE;
   "H" := FALSE;
END_REGION
END_FUNCTION

FUNCTION "Obtem pressao PSF6" : Void   // FC21, LAD
{ S7_Optimized_Access := 'TRUE' }
VERSION : 0.1
   VAR_OUTPUT
      PSF6 : Real;   // Pressão obtida
   END_VAR
   VAR_TEMP
      "Pressao normalizada" : Real;   // Pressão normalizada
   END_VAR
BEGIN

REGION Network 1
   // Normalização do valor de pressão lido do transmissor
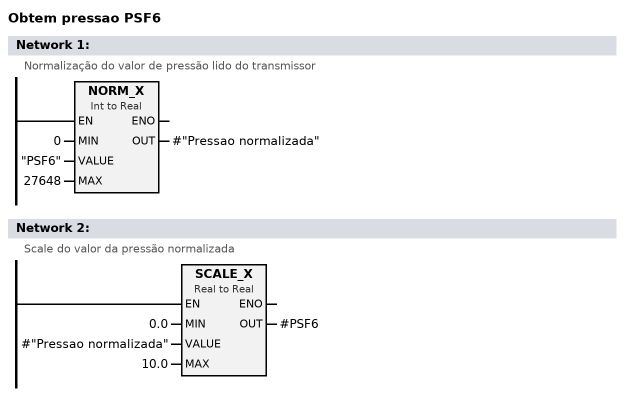
   RUNG wire#powerrail
      { S7_Templates := "[SrcType := Int, DestType := Real]" } Normalize(min := 0, value := "PSF6", max := 27648, out => #"Pressao normalizada")
   END_RUNG
   // the same network as SCL:
   #"Pressao normalizada" := NORM_X(MIN := 0, VALUE := "PSF6", MAX := 27648);
END_REGION

REGION Network 2
   // Scale do valor da pressão normalizada
   RUNG wire#powerrail
      { S7_Templates := "[SrcType := Real, DestType := Real]" } Scale(min := 0.0, value := #"Pressao normalizada", max := 10.0, out => #PSF6)
   END_RUNG
   // the same network as SCL:
   #PSF6 := SCALE_X(MIN := 0.0, VALUE := #"Pressao normalizada", MAX := 10.0);
END_REGION
END_FUNCTION

FUNCTION "Obtem temperatura T" : Void   // FC22, LAD
{ S7_Optimized_Access := 'TRUE' }
VERSION : 0.1
   VAR_OUTPUT
      T : Real;   // Temperatura obtida
   END_VAR
   VAR_TEMP
      "Temperatura normalizada" : Real;   // Temperatura normalizada
   END_VAR
BEGIN

REGION Network 1
   // Normalização do valor de temperatura lido do transmissor
